Fanuc KAREL source: kb00075.KL

-- PROVISIONAL review KL for V770-1; original PC SHA256 dd9361ac7566a91ea61c68d2443e420a98eda0e61af722448c3248e7830ca657
-- Incomplete behavior may be omitted. Consult companion uncertainty JSON. Do not deploy.
PROGRAM KB00075
%NOLOCKGROUP
BEGIN
  -- UNRESOLVED_PC offsets 5-14; opcodes 3F,75
  -- UNRESOLVED_PC offsets 19-28; opcodes 3F,75
  -- UNRESOLVED_PC offsets 33-40; opcodes 9D,23
  -- UNRESOLVED_PC offsets 45-52; opcodes 9D,23
  -- UNRESOLVED_PC offsets 57-89; opcodes 27,22,2A,22,2A,22,22,31
  -- UNRESOLVED_PC offsets 94-98; opcodes 7F
END KB00075
